// LS Electric XG5000 project: 동남108
// PLC NewPLC
// module base 0 slot 0: 입출력 모듈:XBC-DN/DP14E (DC 24V 입력 8점, 트랜지스터 출력 6점)

PROGRAM NewProgram (task: 스캔 프로그램)

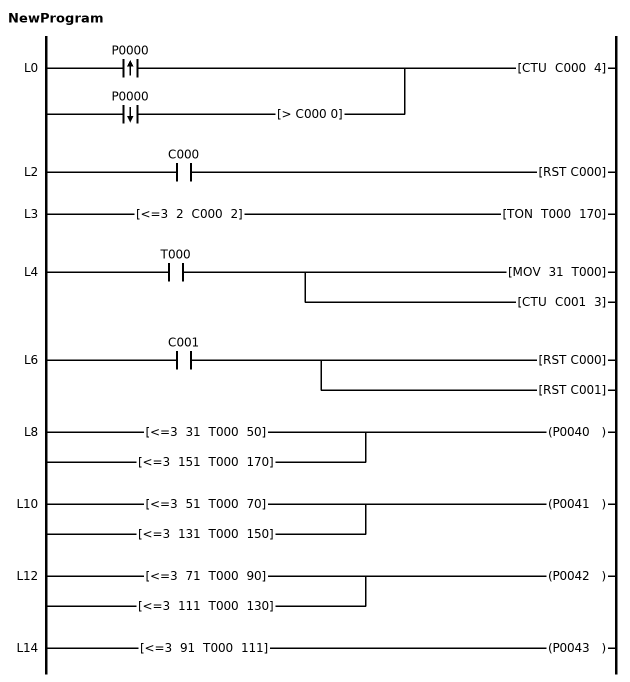
; L0
LOADP     P0000
LOADN     P0000
AND>      C000 0
OR LOAD
CTU       C000 4
; L2
LOAD      C000
RST       C000
; L3
LOAD<=3   2 C000 2
TON       T000 170
; L4
LOAD      T000
MOV       31 T000
CTU       C001 3
; L6
LOAD      C001
RST       C000
RST       C001
; L8
LOAD<=3   31 T000 50
OR<=3     151 T000 170
OUT       P0040
; L10
LOAD<=3   51 T000 70
OR<=3     131 T000 150
OUT       P0041
; L12
LOAD<=3   71 T000 90
OR<=3     111 T000 130
OUT       P0042
; L14
LOAD<=3   91 T000 111
OUT       P0043